FUNCTION_BLOCK FB_MoveFS_Exte
VAR_INPUT
	enable	:BOOL;
	ref		:AXIS_REF;
	jogF	:BOOL;
	jogB	:BOOL;
	Move_Stop:BOOL;
	PosLimit			:BOOL;			(*正极限位信号*)
	NegLimit			:BOOL;			(*负极限位信号*)
	maxDistance			:LREAL;			(*最大行程*)
	Acceleration		:LREAL;
	Deceleration		:LREAL;
	Jerk				:LREAL;
END_VAR
VAR_OUTPUT	
END_VAR
VAR
	MC_Read:MC_ReadStatus;
	MC_ABS:MC_MoveAbsolute;
	MC_REL:MC_MoveRelative;
	MC_Jog:MC_Jog;
	
	MC_ABS1:MC_MoveAbsolute;

	step1,step2,step3		:INT;	
	R_TRIG1,R_TRIG2,R_TRIG3	:R_TRIG;
	R_TRIG_done				:R_TRIG;
	ton_NotMoving			:TON;
	ton_Moving				:TON;
	rel_do					:BOOL;
	abs_do					:BOOL;
	jogF_do					:BOOL;
	jogB_do					:BOOL;
	
	abs_do1    			    :BOOL;
	error					:BOOL;

	MoveAbsolute_Busy		:BOOL;
	MoveConstantVelocity_Busy:BOOL;
	MoveRelative_Busy		:BOOL;
	jog_EN					:BOOL;
	FB_START_r_trig:		R_TRIG;
	start					:BOOL;
	jog_f_trig				:F_TRIG;
	ton_NotMoving_r_trig:Tc2_Standard.R_TRIG;
	Positive_Direction:BOOL;//正向
	Negative_Direction:BOOL;//负向
	
END_VAR
VAR_IN_OUT 
	MoveRelExe					:BOOL;
	MoveAbsExe					:BOOL;
	MoveConstantVelocityExe		:BOOL;//
	Velo						:LREAL;	//mm/s
	TargetRel					:LREAL;//mm
	TargetAbs					:LREAL;//mm
	ConstantVelocityStart		:LREAL;//mm		The position to start moving with a constant velocity
												//      0 < ConstantVelocityStart< ConstanVelocityEnd< RequestedPosition
	ConstanVelocityEnd			:LREAL;//mm		The position to end moving with a constant velocity											
	Done						:BOOL;
	NotMovingTimeOut 			:BOOL;
	SpeedNotReach				:BOOL;
END_VAR

(*********************NOT MOVING TIMEOUT***************************)
FB_START_r_trig(CLK:=jogF OR jogB OR MoveRelExe OR MoveAbsExe OR MoveConstantVelocityExe  , Q=> );
IF FB_START_r_trig.Q THEN 
	start:=TRUE;
END_IF
ton_NotMoving(IN:=Ref.Status.NotMoving AND start  , PT:= T#5S, Q=> , ET=> );
ton_NotMoving_r_trig(CLK:=ton_NotMoving.Q , Q=> );
IF ton_NotMoving_r_trig.Q THEN 
		NotMovingTimeOut:=TRUE;	
END_IF

Call_FB();
JOG();
MoveAbsolute();
MoveConstantVelocity();
MoveRelative();


(*********************error***************************)
IF ton_NotMoving.Q OR error OR SpeedNotReach THEN	
	start:=FALSE;
	error:=FALSE;
	ton_NotMoving(IN:=FALSE);	
	step1:=step2:=step2:=0;	
	MoveRelExe:=FALSE;
	MoveAbsExe:=FALSE;
	MoveConstantVelocityExe:=FALSE;
	Velo:=0;
	TargetAbs:=0;
	TargetRel:=0;
	ConstantVelocityStart:=0;
	ConstanVelocityEnd:=0;
	step1:=step2:=step3:=0;
	R_TRIG1(CLK:=FALSE);
	R_TRIG2(CLK:=FALSE);
	R_TRIG3(CLK:=FALSE);
END_IF

(*********************move done***************************)
IF MoveAbsolute_Busy OR MoveConstantVelocity_Busy OR  MoveRelative_Busy THEN 
	Done:=FALSE;
	jogF:=FALSE;
	jogB:=FALSE;
END_IF

jog_f_trig(CLK:=jogB OR jogF , Q=> );

R_TRIG_done(CLK:=MC_REL.Done OR MC_ABS.Done OR MC_ABS1.Done  OR jog_f_trig.Q OR Move_Stop , Q=> );
IF R_TRIG_done.Q THEN 	
	start:=FALSE;
	R_TRIG_done(CLK:=FALSE);
	NotMovingTimeOut:=FALSE;
	ton_NotMoving(IN:=FALSE);
	step1:=step2:=step3:=0;	
	MoveRelExe:=FALSE;
	MoveAbsExe:=FALSE;
	MoveConstantVelocityExe:=FALSE;
	Velo:=0;
	TargetAbs:=0;
	TargetRel:=0;
	ConstantVelocityStart:=0;
	ConstanVelocityEnd:=0;
	Done:=TRUE ;
END_IF

ACTION Call_FB:
MC_Read(
	Axis:=ref , 
	Enable:=TRUE);
MC_REL(
	Axis:=ref , 
	Execute:=rel_do , 
	Distance:=TargetRel , 
	Velocity:=Velo , 
	Acceleration:=Acceleration , 
	Deceleration:=Deceleration , 
	Jerk:=Jerk , 
	BufferMode:= , 
	Options:= , 
	Done=> , 
	Busy=>MoveRelative_Busy , 
	Active=> , 
	CommandAborted=> , 
	Error=> , 
	ErrorID=> );
	IF MC_REL.Busy THEN 
		rel_do:=FALSE;
		MoveRelExe:=FALSE;
	END_IF
MC_ABS(
	Axis:=ref , 
	Execute:=abs_do , 
	Position:=TargetAbs , 
	Velocity:=Velo , 
	Acceleration:=Acceleration , 
	Deceleration:=Deceleration , 
	Jerk:=Jerk , 
	BufferMode:= , 
	Options:= , 
	Done=> , 
	Busy=>MoveAbsolute_Busy , 
	Active=> , 
	CommandAborted=> , 
	Error=> , 
	ErrorID=> );
	IF MC_ABS.Busy THEN 
		abs_do:=FALSE;
		MoveAbsExe:=FALSE;
	END_IF
MC_Jog(
	Axis:=ref , 
	JogForward:=jogF_do , 
	JogBackwards:=jogB_do , 
	Mode:=MC_JOGMODE_CONTINOUS , 
	Position:= , 
	Velocity:=Velo , 
	Acceleration:=Acceleration , 
	Deceleration:=Deceleration , 
	Jerk:=Jerk , 
	Done=> , 
	Busy=> , 
	Active=> , 
	CommandAborted=> , 
	Error=> , 
	ErrorID=> );
MC_ABS1(
	Axis:=ref , 
	Execute:=abs_do1 , 
	Position:=TargetAbs , 
	Velocity:=Velo , 
	Acceleration:=Acceleration , 
	Deceleration:=Deceleration , 
	Jerk:=Jerk , 
	BufferMode:= , 
	Options:= , 
	Done=> , 
	Busy=> , 
	Active=> , 
	CommandAborted=> , 
	Error=> , 
	ErrorID=> );
	IF MC_ABS1.Busy THEN 
		abs_do1:=FALSE;
		MoveConstantVelocityExe:=FALSE;
	END_IF
END_ACTION

ACTION JOG:
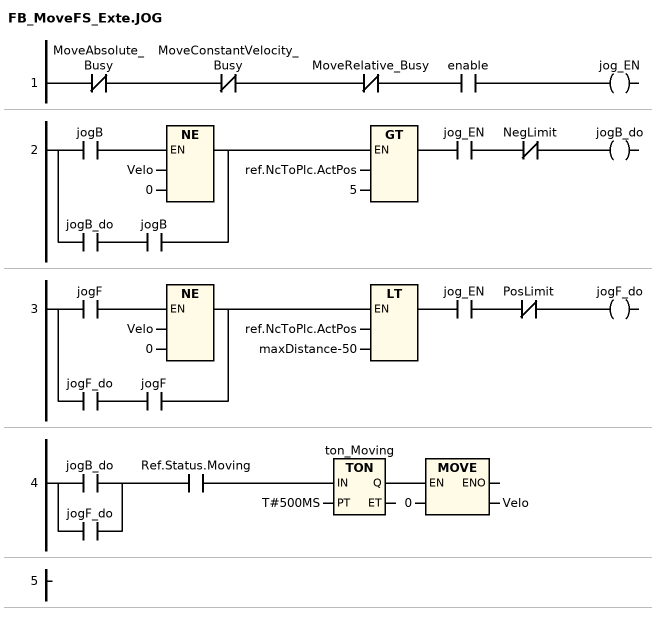
// NETWORK 1
jog_EN := NOT MoveAbsolute_Busy AND NOT MoveConstantVelocity_Busy AND NOT MoveRelative_Busy AND enable;

// NETWORK 2
jogB_do := ((jogB AND Velo <> 0 OR jogB_do AND jogB) AND ref.NcToPlc.ActPos > 5) AND jog_EN AND NOT NegLimit;

// NETWORK 3
jogF_do := ((jogF AND Velo <> 0 OR jogF_do AND jogF) AND ref.NcToPlc.ActPos < (maxDistance-50)) AND jog_EN AND NOT PosLimit;

// NETWORK 4
ton_Moving(IN := (jogB_do OR jogF_do) AND Ref.Status.Moving, PT := T#500MS); // TON
IF ton_Moving.Q THEN Velo := 0; END_IF

// NETWORK 5
END_ACTION

ACTION MoveAbsolute:
(****************ABS********************)
R_TRIG2(CLK:=MoveAbsExe AND Ref.Status.NotMoving AND enable   , Q=> );

CASE step2 OF 
	0:				
		IF R_TRIG2.Q THEN 
			R_TRIG2(CLK:=FALSE);			
			MoveAbsExe:=FALSE;
			step2:=1;
		END_IF
	1:	
		IF   Velo<>0 THEN 		
			abs_do:=TRUE;
			step2:=2;
		END_IF
	2:
		IF MC_ABS.Busy THEN 
			abs_do:=FALSE;								
			step2 :=0;
		END_IF	
END_CASE


IF  MoveAbsolute_Busy THEN 
	MoveRelExe:=FALSE;
	MoveConstantVelocityExe:=FALSE;
END_IF
END_ACTION

ACTION MoveConstantVelocity:
(****************MoveConstantVelocity********************)
R_TRIG3(CLK:=MoveConstantVelocityExe AND Ref.Status.NotMoving AND enable  , Q=> );
CASE step3 OF 
	0:				
		IF R_TRIG3.Q THEN 
			R_TRIG3(CLK:=FALSE);
			abs_do1:=FALSE;		
			MoveConstantVelocityExe:=FALSE;
			step3:=1;
		END_IF
	1:	//
		IF   Velo<>0 THEN 		
			abs_do1:=TRUE;
			step3:=2;
		END_IF
		
	2:	//启动第二段，匀速段,增加到达位置时速度判断
		IF ConstanVelocityEnd>ConstantVelocityStart THEN 
			Positive_Direction:=TRUE;
			Negative_Direction:=FALSE;
		ELSE
			Positive_Direction:=FALSE;
			Negative_Direction:=TRUE;	
		END_IF

			
		IF 	(Positive_Direction AND ref.NcToPlc.ActPos>=ConstantVelocityStart ) OR 
			(Negative_Direction AND ref.NcToPlc.ActPos<=ConstantVelocityStart ) THEN 
			
			 IF ABS(ABS(ref.NcToPlc.ActVelo)-Velo)<=30 THEN
				step3 :=3;
			 ELSE  
				step3 :=5;
			 END_IF
			
		END_IF
	3://满足第一段加速,检测减速度
		IF 	ABS(ref.NcToPlc.ActPos-ConstanVelocityEnd)<=30  THEN 
			IF ABS(ABS(ref.NcToPlc.ActVelo)-Velo)<=30 THEN
				step3 :=0;
			 ELSE  
				step3 :=5;
			 END_IF  
		END_IF	 
	5://ERROR
		SpeedNotReach:=TRUE;
		step3 :=0;
		
END_CASE
MoveConstantVelocity_Busy:=MC_ABS1.Busy ;

IF MoveConstantVelocity_Busy THEN 
	MoveRelExe:=FALSE;
	MoveAbsExe:=FALSE;
END_IF
END_ACTION

ACTION MoveRelative:
(****************Rel********************)
R_TRIG1(CLK:=MoveRelExe AND Ref.Status.NotMoving AND enable  , Q=> );
CASE step1 OF 
	0:				
		IF R_TRIG1.Q THEN 
			R_TRIG1(CLK:=FALSE);
			MoveRelExe:=FALSE;
			step1:=1;
		END_IF
	1:	
		IF TargetRel <>0 AND Velo<>0 THEN 		
			rel_do:=TRUE;
			step1:=2;
		END_IF
	2:
		IF MC_REL.Busy THEN 
			rel_do:=FALSE;								
			step1 :=0;
		END_IF	
END_CASE

IF MoveRelative_Busy THEN 
	MoveAbsExe:=FALSE;
	MoveConstantVelocityExe:=FALSE;
END_IF
END_ACTION

END_FUNCTION_BLOCK

(* stored: Version 1.1.0.1, ProductVersion 3.1.4024.11
   POU FB_MoveFS_Exte: Id {841919f6-7681-4bd7-b0bb-d66d9f1c2a4c}, SpecialFunc None
   Action Call_FB: Id {fb9b0b54-df4a-4859-b1af-168f1664cc5d}
   Action JOG: Id {3a0be207-1e4a-45ed-9718-487ac6aa30f4}
   Action MoveAbsolute: Id {e097955a-8fd0-4833-9aa8-204e160a0d21}
   Action MoveConstantVelocity: Id {fefa3c2c-45e9-4ded-a8c8-67f3c5082895}
   Action MoveRelative: Id {bab86dd1-6c12-4e48-87fd-8aa89432f826} *)
